# EPICS autosave request: iocBoot/gmca_23i_ioc2/dbSave/axs1.req
%
% BURT Request File
%
% AXIS
%

% RO $(AXS1):ActPos
$(AXS1):ActPos.EGU
$(AXS1):ActPos.DESC

$(AXS1):RqsPos
$(AXS1):RqsPos.EGU
$(AXS1):RqsPos.DESC
$(AXS1):RqsPos.HOPR
$(AXS1):RqsPos.LOPR
$(AXS1):RqsPos.DRVH
$(AXS1):RqsPos.DRVL

$(AXS1):RqsBkl
$(AXS1):RqsBkl.EGU
$(AXS1):RqsBkl.DESC

$(AXS1):RqsPosInc
$(AXS1):MemPos
